TEXTLIST TL_BitConventer
  0 = 'Choose'
  1 = '12-bit'
  2 = '16-bit'
   = ''
END_TEXTLIST

(* stored: Version 1.1.0.1, ProductVersion 3.1.4020.3
   TextList TL_BitConventer: Id {efaea4f7-3a25-4410-8735-39c50bde1c76} *)
